FUNCTION_BLOCK TcoContextTest EXTENDS TcoContext
VAR
	_CallMyPlcInstance 		:	BOOL := FALSE;
	_startCycles			:	ULINT;
	_endCycles				:	ULINT;	
	_mainCycles				:	ULINT;
	_TcoObjectTest_A		:	TcoObjectTest(THIS^);
	_TcoObjectTest_B		:	TcoObjectTest(THIS^);
	_MyIdentity				:	ULINT;	
END_VAR

IF THIS^._CallMyPlcInstance THEN
	THIS^.Run();
END_IF

{attribute 'TcRpcEnable'}
METHOD INTERNAL CallMainFromUnitTest
THIS^.Main();
END_METHOD

{attribute 'TcRpcEnable'}
METHOD INTERNAL CallRunFromUnitTest
THIS^.Run();
END_METHOD

{attribute 'TcRpcEnable'}
METHOD INTERNAL ContextClose
SUPER^.Close();
END_METHOD

{attribute 'TcRpcEnable'}
METHOD INTERNAL ContextOpen
SUPER^.Open();
END_METHOD

METHOD PROTECTED  Main
_mainCycles := _mainCycles + 1;

_MyIdentity	:= THIS^.Identity;
END_METHOD

{attribute 'TcRpcEnable'}
METHOD INTERNAL ReadOutCycleCounters
_startCycles		:=		THIS^.StartCycleCount;
_endCycles			:=		THIS^.EndCycleCount;

_MyIdentity			:= 		THIS^.Identity;
END_METHOD

END_FUNCTION_BLOCK

(* stored: Version 1.1.0.1, ProductVersion 3.1.4024.6
   POU TcoContextTest: Id {6642835d-5414-4760-aac1-4c8cef083deb}, SpecialFunc None
   Method CallMainFromUnitTest: Id {9c9d295d-40fb-48af-adaf-5d210f5656a3}
   Method CallRunFromUnitTest: Id {06319017-0b6a-4225-bce8-de1fd8b0ed0e}
   Method ContextClose: Id {4adc0216-d7dc-47d4-a216-4cfc4c14ed41}
   Method ContextOpen: Id {65cd14ad-eb62-4d0c-8ca2-8e3c5c9380bf}
   Method Main: Id {76d8f63c-d45d-4de4-ad73-4298aca95aa1}
   Method ReadOutCycleCounters: Id {3ce97aaa-6bf5-4a06-9e7c-0d88acee2466} *)
